{attribute 'linkalways'} 
{attribute 'no_explicit_call' := 'This FB is a CLASS and must be accessed using methods or properties'}
{attribute 'enable_dynamic_creation'}
FUNCTION_BLOCK _ETcVnSignedNormalization EXTENDS EnumDatatypeBase
VAR
	localData : ETcVnSignedNormalization;
	activeData : REFERENCE TO ETcVnSignedNormalization;
	enumBaseDatatype : _INT(localData);
END_VAR

METHOD PRIVATE AddLocalEnumeration
VAR_INPUT
	Enumeration : T_MAXSTRING;
	Value : ETcVnSignedNormalization;
END_VAR
AddEnumeration(Enumeration, Value);
END_METHOD

PROPERTY PUBLIC Address : PVOID
GET
Address := ADR(activeData);
END_GET
END_PROPERTY

METHOD PUBLIC ClearReference
VAR_INPUT
END_VAR
activeData REF= localData;
SetBaseDatatypeReference();
END_METHOD

METHOD PUBLIC Clone : I_Datatype
VAR
    pClone : POINTER TO _ETcVnSignedNormalization;
END_VAR
pClone := __NEW(_ETcVnSignedNormalization(InitialValue := Value));
Clone := pClone^;
END_METHOD

METHOD FB_init : BOOL
VAR_INPUT
	bInitRetains : BOOL; // if TRUE, the retain variables are initialized (warm start / cold start)
	bInCopyCode : BOOL;  // if TRUE, the instance afterwards gets moved into the copy code (online change)
	InitialValue : ETcVnSignedNormalization;
END_VAR
localData := InitialValue;
AddBaseDatatype(enumBaseDatatype);
ClearReference();

AddLocalEnumeration('TCVN_SN_FIX_ZERO', ETcVnSignedNormalization.TCVN_SN_FIX_ZERO);
AddLocalEnumeration('TCVN_SN_FULL_SCALE', ETcVnSignedNormalization.TCVN_SN_FULL_SCALE);
END_METHOD

PROPERTY PUBLIC Identifier : T_MAXSTRING
GET
Identifier := 'ETcVnSignedNormalization';
END_GET
END_PROPERTY

METHOD IsEnumeratorValueEqual : BOOL
VAR_INPUT
	Enumerator : I_KeyValueForwardEnumerator;
END_VAR
VAR
	storedValue : ETcVnSignedNormalization;
END_VAR
IF NOT Enumerator.TryGet(storedValue) THEN
	RETURN;
END_IF

IsEnumeratorValueEqual := storedValue = activeData;
END_METHOD

METHOD PUBLIC MakeReferenceTo
VAR_INPUT
	ReferenceTarget : REFERENCE TO ETcVnSignedNormalization;
END_VAR
activeData REF= ReferenceTarget;
SetBaseDatatypeReference();
END_METHOD

METHOD PROTECTED SetBaseDatatypeReference
VAR_INPUT
END_VAR
enumBaseDatatype.MakeReferenceTo(activeData);
END_METHOD

PROPERTY PUBLIC Size : UDINT
GET
Size := SIZEOF(activeData);
END_GET
END_PROPERTY

METHOD TryMakeReferenceTo : BOOL
VAR_INPUT
	Target : I_Datatype;
END_VAR
VAR
	targetAsEnum : I_EnumDatatype;
	pTargetData : POINTER TO ETcVnSignedNormalization;
END_VAR
IF NOT Target.TryResolveAsEnumDatatype(targetAsEnum) THEN
	RETURN;
END_IF

IF targetAsEnum.Identifier <> Identifier THEN
	RETURN;
END_IF

pTargetData := Target.Address;
activeData REF= pTargetData^;
SetBaseDatatypeReference();
TryMakeReferenceTo := TRUE;
END_METHOD

PROPERTY PUBLIC Value : ETcVnSignedNormalization
GET
Value := activeData;
END_GET
SET
activeData := Value;
END_SET
END_PROPERTY

END_FUNCTION_BLOCK

(* stored: Version 1.1.0.1
   POU _ETcVnSignedNormalization: Id {7785e906-d6bb-4797-aab7-4acc288328e7}, SpecialFunc None
   Folder Constructor: Id {83e0747b-8be3-41a8-94e0-fe52836a8312}
   Folder Private: Id {6f4313dd-ee08-4c47-8a17-64a68d2b5ecf}
   Folder Protected: Id {09597106-fd8d-4352-b1c5-2511b5dc58c8}
   Method AddLocalEnumeration: Id {bef39e62-2dc3-4247-872d-5e577ed775f1}
   Property Address: Id {be479d87-16c8-4867-9237-430067b8df01}
   Get Get: Id {bb36820e-da9c-4791-8d83-aa812d58bff8}
   Method ClearReference: Id {04b36882-488e-4a94-8e98-f47929dd7c52}
   Method Clone: Id {fc6b1644-ce02-46b5-8a25-6dfd76edc281}
   Method FB_init: Id {b98a0632-db95-4c71-b446-0ce675666ab9}
   Property Identifier: Id {93fefc0a-45c9-4fa0-b41b-091b11f8214f}
   Get Get: Id {df86a2da-e34e-4685-9700-2fbd05e25a0e}
   Method IsEnumeratorValueEqual: Id {2f1d1de3-1671-4bb8-8dd9-d373abd947cc}
   Method MakeReferenceTo: Id {bf8f37ea-c70b-4cff-ac8d-f02ede94421f}
   Method SetBaseDatatypeReference: Id {1a6fa5ed-7020-4684-a671-6ad25e96ad73}
   Property Size: Id {db60c148-abed-4db7-b8c6-05269c6936e6}
   Get Get: Id {0e620065-baa2-4ff5-98e8-eb30e4748a9d}
   Method TryMakeReferenceTo: Id {5c485ff2-96fe-4500-b46f-1b952c1c19e8}
   Property Value: Id {74036c7d-1239-4ae4-9361-5924573379c6}
   Get Get: Id {92c3801f-3a96-4d1b-8e7e-1a2d127892c3}
   Set Set: Id {6c3ca591-e1ae-4e90-a6f1-bfffc7a82461} *)
